(*
Purpose:     Base for Devices 
             FD_Device includes standard properties and standard methodes
*)

FUNCTION_BLOCK ABSTRACT FD_Device EXTENDS FB_Base IMPLEMENTS ITF_Device, ITF_Owner
VAR_INPUT
END_VAR
VAR_OUTPUT
END_VAR
VAR
	itfDeviceRegister									: ITF_Owner;
	aitfChilds												: ARRAY [1..GVL_Core.C_MaxChild] OF ITF_Device;     // Registered child devices
	uiChildsCount											: UINT := 0;                                       	// Number of registered child devices
	
	eMode															: E_Mode;
	uiSequenceID          						: UINT;
	uiNextStep      									: UINT;
	                									
	bHomed          									: BOOL;
	bReady          									: BOOL;
	                									
	bSequenceBusy   									: BOOL;
	bSequenceDone   									: BOOL;
	                									
	bHold           									: BOOL;
	bAbort          									: BOOL;

END_Var

VAR CONSTANT
 //***********************************************************  CONSTANT  C_SeqStep
 C_SeqStep_Idle                   	: UINT :=   0;                    
 C_SeqStep_Start                  	: UINT :=   1;                    
 C_SeqStep_Done                 		: UINT :=   2;  									              
 C_SeqStep_Error                		: UINT :=   3;  									
 C_SeqStep_Abort                		: UINT :=   4;  									 
 C_SeqStep_Undefined            		: UINT :=   5;  							
		
END_VAR


SUPER^();
IF NOT Enable THEN RETURN; END_IF;

IF bError
	THEN
  	mStop(TRUE);
    RETURN;
END_IF;

IF bSequenceBusy THEN mSequence(TRUE); END_IF;

//FB_Init ist immer implizit verfügbar und wird primär für die Initialisierung verwendet.
//Der Rückgabewert wird nicht ausgewertet. Für gezielte Einflussnahme können Sie
//die Methoden explizit deklarieren und darin mit dem Standard-Initialisierungscode 
//zusätzlichen Code bereitstellen. Sie können den Rückgabewert auswerten.
METHOD FB_Init: BOOL
VAR_INPUT    
	bInitRetains					: BOOL; 					// TRUE: Die Retain-Variablen werden initialisiert (Reset warm / Reset kalt)    
	bInCopyCode						: BOOL;  					// TRUE: Die Instanz wird danach in den Kopiercode kopiert (Online-Change)
	
	I_Name                : STRING;         //  Name
	I_ID                  : UINT;           // ID
  I_itfOwner					  : ITF_Owner;      // owner 
END_VAR

IF I_itfOwner <>0
	THEN
		itfDeviceRegister 	:= I_itfOwner;
		itfDeviceRegister.mRegisterChild(THIS^);
END_IF

// Default sequence state
SequenceID 							:= C_SeqStep_Idle;

bSequenceBusy 					:= FALSE;
bSequenceDone 					:= FALSE;
              					
bReady 									:= FALSE;
bHomed									:= FALSE;
bAbort 									:= FALSE;
bHold 									:= FALSE;
END_METHOD

PROPERTY Homed : BOOL
GET
Homed := bHomed;
END_GET
SET
bHomed := Homed;
END_SET
END_PROPERTY

METHOD mAbort : E_CmdState
VAR_INPUT
	I_bExecute : BOOL;
END_VAR
IF NOT I_bExecute 
	THEN
    mAbort     := E_CmdState.Idle;
    RETURN;
END_IF

bAbort         := TRUE;
bSequenceBusy  := FALSE;
bSequenceDone  := FALSE;

SequenceID     := C_SeqStep_Idle;

mStop(TRUE);

mAbort := E_CmdState.Busy;
END_METHOD

METHOD mAutomatic: E_CmdState
VAR_INPUT
	I_bExecute : BOOL;
END_VAR
// No command requested.
IF NOT I_bExecute THEN
    mAutomatic := E_CmdState.Idle;
    RETURN;
END_IF

// Device disabled / not initialized / not homming
IF NOT Enable OR NOT bHomed
	THEN
    mAutomatic := E_CmdState.NotReady;
    RETURN;
END_IF

// Device is in error state.
IF bError 
	THEN
		SequenceID := C_SeqStep_Error;
    mAutomatic := E_CmdState.Error;
    RETURN;
END_IF

Mode := E_Mode.Auto;

// Start sequence execution.
bSequenceBusy 	:= TRUE;
bSequenceDone 	:= FALSE;
SequenceID     	:= C_SeqStep_Start;
mAutomatic 			:= E_CmdState.Busy;
END_METHOD

METHOD mDone : E_CmdState
VAR_INPUT
END_VAR
(*


*)
IF bError
  THEN 
		mDone :=  E_CmdState.Failed;	
  ELSE 
		mDone :=  E_CmdState.Succeeded;
END_IF

bSequenceBusy := FALSE;
bSequenceDone := TRUE;
SequenceID := C_SeqStep_Idle;
END_METHOD

METHOD mHold : E_CmdState
VAR_INPUT
	I_bExecute : BOOL;
END_VAR

IF NOT I_bExecute 
	THEN
    mHold := E_CmdState.Idle;
    RETURN;
END_IF

bHold := TRUE;
bSequenceBusy := FALSE;
mHold := E_CmdState.Hold;
END_METHOD

METHOD mHome : E_CmdState
VAR_INPUT
	I_bExecute : BOOL;
END_VAR
// No command requested.
IF NOT I_bExecute 
	THEN
    mHome := E_CmdState.Idle;
    RETURN;
END_IF

// Device disabled.
IF NOT Enable 
	THEN
    mHome := E_CmdState.NotReady;
    RETURN;
END_IF

// Device in error.
IF Error 
	THEN
    mHome := E_CmdState.Error;
    RETURN;
END_IF
// Device already running another sequence.
IF SequenceBusy 
	THEN
    mHome := E_CmdState.Busy;
    RETURN;
END_IF

// Start local homing sequence.
Mode := E_Mode.Homing;

SequenceBusy := TRUE;
SequenceDone := FALSE;

Homed := FALSE;
Ready := FALSE;

SequenceID := C_SeqStep_Start;

mHome := E_CmdState.Busy;
END_METHOD

PROPERTY Mode : E_Mode
GET
Mode := eMode;
END_GET
SET
eMode := Mode;
END_SET
END_PROPERTY

METHOD mRegisterChild : BOOL
VAR_INPUT
	I_itfChild        : ITF_Device;
END_VAR

VAR 
	L_Itf_ChildDevice : ITF_Device := 0;
END_VAR


IF __QUERYINTERFACE (I_itfChild, L_Itf_ChildDevice)
	THEN 
		IF uiChildsCount < GVL_Core.C_MaxChild
			THEN 
				uiChildsCount 								:= uiChildsCount +1;	
				aitfChilds[uiChildsCount] 		:= L_Itf_ChildDevice;
		END_IF
END_IF
END_METHOD

METHOD mRelease : E_CmdState
VAR_INPUT
	I_bExecute : BOOL;
END_VAR

IF NOT I_bExecute 
	THEN
    mRelease 	:= E_CmdState.Idle;
    RETURN;
END_IF

bHold    			:= FALSE;
bAbort   			:= FALSE;
         			
mRelease 			:= E_CmdState.Busy;
END_METHOD

METHOD mReset : BOOL
VAR_INPUT

END_VAR

SUPER^.mReset();
END_METHOD

METHOD mSequence : E_CmdState
VAR_INPUT
	I_bExecute : BOOL;
END_VAR

IF NOT I_bExecute 
	THEN
    mSequence := E_CmdState.Idle;
    RETURN;
END_IF

IF bError 
	THEN
		SequenceID := C_SeqStep_Error;
    mSequence  := E_CmdState.Error;
    RETURN;
END_IF

// Allows for a clean stop of a sequence.
IF bAbort 
	THEN
    SequenceID := C_SeqStep_Abort;
    mSequence := E_CmdState.Aborted;
    RETURN;
END_IF

//Hold allows for pausing without losing the SequenceID.
IF bHold 
	THEN
    mSequence := E_CmdState.Busy;
    RETURN;
END_IF

bSequenceBusy := TRUE;
bSequenceDone := FALSE;

mSequence := E_CmdState.Busy;
END_METHOD

METHOD mService : E_CmdState
VAR_INPUT
	I_bExecute : BOOL;
END_VAR
IF NOT I_bExecute 
	THEN
    mService := E_CmdState.Idle;
    RETURN;
END_IF

Mode := E_Mode.Service;
bSequenceBusy := FALSE;
bSequenceDone := FALSE;

mService := E_CmdState.Busy;
END_METHOD

METHOD mSetChildOpMode : BOOL
VAR_INPUT
	I_eSetChilds  : E_SetChild;
END_VAR
VAR
	L_uiIndex			: UINT;
END_VAR

FOR L_uiIndex := 1 TO uiChildsCount DO
	CASE I_eSetChilds OF
		E_SetChild.None					: ;
		E_SetChild.Enable				:	aitfChilds[L_uiIndex].Enable:= Enable; 
		E_SetChild.Reset 				: aitfChilds[L_uiIndex].mReset();	
		E_SetChild.Abort				:	aitfChilds[L_uiIndex].mAbort(TRUE);
//		E_SetChild.ClearError		:	aitfChilds[L_uiIndex].mError(TRUE);
		E_SetChild.EStop				:	aitfChilds[L_uiIndex].mStop(TRUE);
		E_SetChild.Auto					: aitfChilds[L_uiIndex].mAutomatic(TRUE);
		E_SetChild.Servic				: aitfChilds[L_uiIndex].mService(TRUE);
		E_SetChild.Home					: aitfChilds[L_uiIndex].mHome(TRUE);
		E_SetChild.Release			: aitfChilds[L_uiIndex].mRelease(TRUE);
	END_CASE
END_FOR
END_METHOD

METHOD mStop : E_CmdState
VAR_INPUT
	I_bExecute : BOOL;
END_VAR
IF NOT I_bExecute 
	THEN
  	mStop 			:= E_CmdState.Idle;
    RETURN;
END_IF

Mode := E_Mode.Error;

bBusy 					:= FALSE;
bDone 					:= FALSE;
bSequenceBusy 	:= FALSE;
bSequenceDone 	:= FALSE;

SequenceID     	:= C_SeqStep_Idle;
mStop 					:= E_CmdState.Succeeded;
END_METHOD

PROPERTY Ready : BOOL
GET
Ready := bReady;
END_GET
SET
bReady := Ready;
END_SET
END_PROPERTY

PROPERTY SequenceBusy : BOOL
GET
SequenceBusy := bSequenceBusy;
END_GET
SET
bSequenceBusy := SequenceBusy;
END_SET
END_PROPERTY

PROPERTY SequenceDone : BOOL
GET
SequenceDone := bSequenceDone ;
END_GET
SET
bSequenceDone := SequenceDone ;
END_SET
END_PROPERTY

PROPERTY SequenceID : UINT
GET
SequenceID := uiSequenceID;
END_GET
SET
uiSequenceID := SequenceID;
END_SET
END_PROPERTY

END_FUNCTION_BLOCK

(* stored: Version 1.1.0.1, ProductVersion 3.1.4026.18
   POU FD_Device: Id {571b9eee-9c23-4a84-ac31-37e95ea393f3}, SpecialFunc None
   Folder 01 Properties: Id {2ade4f6f-4d16-4ebd-be39-d23d9d34597f}
   Folder 02 Methodes: Id {34903398-ece8-40e6-8ccd-c04371e5f652}
   Folder _SetChild: Id {1eae8e4b-4066-46b8-876f-e8b83ce863d5}
   Folder OpMode: Id {d1c9d0a0-c08d-4381-9e61-4553d39a7da0}
   Method FB_Init: Id {7fd52798-a9d4-47c6-81da-6550d3521908}
   Property Homed: Id {f8978509-4b98-4bbf-bb6e-7234335367a3}
   Get Get: Id {e0ded4dc-1f5b-4e59-9a3a-0f03e39f212d}
   Set Set: Id {635d479a-5bb6-4b03-8771-b1189ad6129d}
   Method mAbort: Id {37a9e74e-74b2-46c6-b456-57916c5147b4}
   Method mAutomatic: Id {1893a5c2-c84c-454f-8d17-e1b9361eb323}
   Method mDone: Id {de0d20d5-1293-42e2-9278-5a9f25f8ea1d}
   Method mHold: Id {f28f09b1-dbdb-4357-9970-1dd737918a37}
   Method mHome: Id {d161db35-b843-4f4b-9979-193f62066daf}
   Property Mode: Id {e3629892-5ebc-4865-8c65-e29d8930dd33}
   Get Get: Id {5bea1d50-c46c-45c6-97f9-e0b4c5cb818c}
   Set Set: Id {39899aae-4e47-4f77-9b37-e0404462fc6b}
   Method mRegisterChild: Id {a500345d-fc2f-4016-bc40-685c8cf16433}
   Method mRelease: Id {e5842ae1-3411-4eb3-97f0-f3398dbccc11}
   Method mReset: Id {65c3f427-09f3-4c2e-9a66-023cec950cf8}
   Method mSequence: Id {ceec0fba-774c-4026-a416-40592d0b39fe}
   Method mService: Id {59a6f5d6-c772-4191-9bcd-24619a63d134}
   Method mSetChildOpMode: Id {dc18dc8c-5754-40d9-9782-aaae2d87f285}
   Method mStop: Id {7e87bb71-0efa-4d7e-ad01-108cb981aa4c}
   Property Ready: Id {218dca75-2ad9-4843-895f-98e750b75e82}
   Get Get: Id {c16d7636-076a-4981-b7a2-fdd91a84d8df}
   Set Set: Id {ee2a586a-beb7-40b6-8826-ad20aa51af67}
   Property SequenceBusy: Id {acf8dd9e-e59e-43d4-8448-a8432c8b8763}
   Get Get: Id {82ab2c7e-99d0-4060-b5b0-1004872311c4}
   Set Set: Id {538c2dd9-9c8d-471a-a0b5-e70154b9658b}
   Property SequenceDone: Id {6f56f0f8-8c2c-4ff8-8647-b1bcdd96766c}
   Get Get: Id {5a241586-5193-4d99-a720-c4e3f2407b59}
   Set Set: Id {ec87f0f2-2027-4b1e-8eec-2cba17ce8e0b}
   Property SequenceID: Id {aeb45a97-1e41-41aa-8b62-964327e6da6d}
   Get Get: Id {bb3578c9-6043-4cb7-9716-3ab8113875e4}
   Set Set: Id {9c7119be-f35a-49ff-9269-c1873d8cd6b4} *)
